(* PLC project SafeLOGIC-1, BrAutomation SafeDESIGNER  4.2.2.18 *)
(* stored: companyURL http://www.br-automation.com, creationDateTime Fri Feb 10 15:48:36 2017 *)

PROGRAM Main

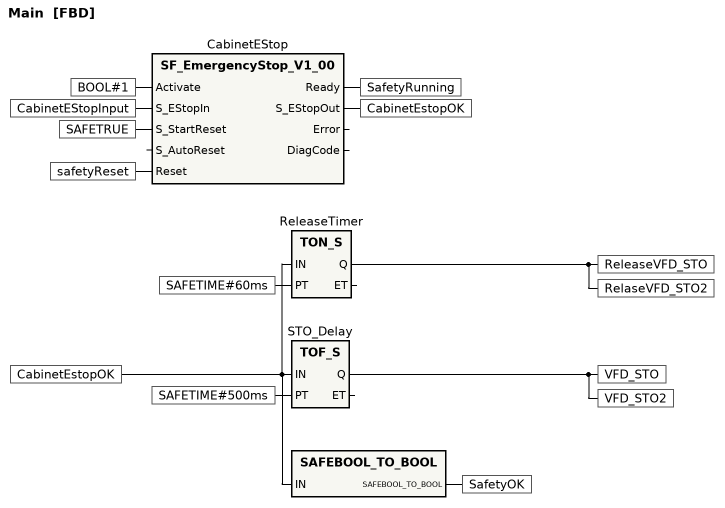
(* FBD diagram, written out as Structured Text *)
CabinetEStop(Activate := BOOL#1, S_EStopIn := CabinetEStopInput, S_StartReset := SAFETRUE, Reset := safetyReset);
CabinetEstopOK := CabinetEStop.S_EStopOut;
SafetyRunning := CabinetEStop.Ready;
SafetyOK := SAFEBOOL_TO_BOOL(CabinetEstopOK);
STO_Delay(IN := CabinetEstopOK, PT := SAFETIME#500ms);
VFD_STO := STO_Delay.Q;
VFD_STO2 := STO_Delay.Q;
ReleaseTimer(IN := CabinetEstopOK, PT := SAFETIME#60ms);
RelaseVFD_STO2 := ReleaseTimer.Q;
ReleaseVFD_STO := ReleaseTimer.Q;
END_PROGRAM
